PROGRAM POU
VAR
END_VAR

END_PROGRAM

(* stored: Version 1.1.0.1, ProductVersion 3.1.4024.13
   POU POU: Id {85d05c48-c160-4e94-91c4-02923575af19}, SpecialFunc None *)
